{attribute 'Tc2GvlVarNames'}
{attribute 'strict'}
TYPE E_XmlVariableType :
(
	eXmlSSMR := 1,
	eXmlSSUR := 2,
	eXmlSSER := 3,
	eXmlProductRecipe := 4
);
END_TYPE

(* stored: Version 1.1.0.1, ProductVersion 3.1.4024.12
   DUT E_XmlVariableType: Id {c46dfe58-2ff6-422a-992f-dbb2d19b6964} *)
